// TIA Portal project "Проект3" (V14)

(* hardware
DEVICE "S7300/ET200M station_1"  S7-300 station
   slot 0: "Профильная шина_0"  Rail  6ES7 390-1***0-0AA0
   slot 2: "PLC_1"  CPU 315-2 PN/DP  6ES7 315-2EH14-0AB0  V3.2
      slot 2: "Интерфейс PROFINET_1"  PN-IO
         slot 1: "Порт_1"  Port
         slot 2: "Порт_2"  Port
   slot 4: "DI 32x24 В пост. тока_1"  DI32 x 24VDC  6ES7 321-1BL00-0AA0
   slot 5: "DO 16x24 В пост. тока/0,5 А_1"  DO16 x 24VDC / 0.5A  6ES7 322-1BH01-0AA0
   slot 6: "AI 8x12 бит_1"  AI8 x 12 bits  6ES7 331-7KF02-0AB0
*)

// ===== PLC "PLC_1"  CPU 315-2 PN/DP =====

VAR_GLOBAL   // PLC tag table "Стандартная таблица переменных"
   "Input_1" AT %I0.0 : Bool;
   "Input_2" AT %I0.1 : Bool;
   "Input_3" AT %I0.2 : Bool;
   "Input_4" AT %I0.3 : Bool;
   "Input_5" AT %I0.4 : Bool;
   "Input_6" AT %I0.5 : Bool;
   "Input_7" AT %I0.6 : Bool;
   "Input_8" AT %I0.7 : Bool;
   "Input_9" AT %I1.0 : Bool;
   "Input_10" AT %I1.1 : Bool;
   "Input_11" AT %I1.2 : Bool;
   "Input_12" AT %I1.3 : Bool;
   "Input_13" AT %I1.4 : Bool;
   "Input_14" AT %I1.5 : Bool;
   "Input_15" AT %I1.6 : Bool;
   "Input_16" AT %I1.7 : Bool;
   "Output_1" AT %Q4.0 : Bool;
   "Output_2" AT %Q4.1 : Bool;
   "Output_3" AT %Q4.2 : Bool;
   "Output_4" AT %Q4.3 : Bool;
   "Output_5" AT %Q4.4 : Bool;
   "Output_6" AT %Q4.5 : Bool;
   "Output_7" AT %Q4.6 : Bool;
   "Output_8" AT %Q4.7 : Bool;
   "Output_9" AT %Q5.0 : Bool;
   "Output_10" AT %Q5.1 : Bool;
   "Output_11" AT %Q5.2 : Bool;
   "Output_12" AT %Q5.3 : Bool;
   "Output_13" AT %Q5.4 : Bool;
   "Output_14" AT %Q5.5 : Bool;
   "Output_15" AT %Q5.6 : Bool;
   "Output_16" AT %Q5.7 : Bool;
   "Tag_1" AT %IW0 : Word;
   "Tag_2" AT %IB0 : Byte;
   "Tag_3" AT %IB1 : Byte;
   "Tag_4" AT %QB4 : Byte;
   "Tag_5" AT %QB5 : Byte;
   "Tag_6" AT %IW288 : Int;
   "Tag_7" AT %M0.1 : Bool;
   "Tag_8" AT %MW1 : Word;
   "Tag_9" AT %MW3 : Word;
   "Tag_10" AT %MD4 : Real;
   "Tag_11" AT %IW290 : Int;
   "Tag_12" AT %IW292 : Int;
   "Tag_13" AT %MW10 : Int;
   "Tag_14" AT %MD20 : Real;
   "Tag_15" AT %MW40 : Word;
   "Tag_16" AT %M0.0 : Bool;
   "Tag_17" AT %IW296 : Int;
   "Tag_18" AT %IW298 : Int;
   "Tag_19" AT %MD30 : Real;
   "Tag_20" AT %QD0 : Real;
END_VAR

DATA_BLOCK "DB_1"   // DB1
{ S7_Optimized_Access := 'FALSE' }
VERSION : 0.1
   VAR
      "Q4.0" : Bool;
      "Q4.1" : Bool;
      "Q4.2" : Bool;
      "Q4.3" : Bool;
      "Q4.4" : Bool;
      "Q4.5" : Bool;
      "Q4.6" : Bool;
      "Q4.7" : Bool;
      "Q5.0" : Bool;
      "Q5.1" : Bool;
      "Q5.2" : Bool;
      "Q5.3" : Bool;
      "Q5.4" : Bool;
      "Q5.5" : Bool;
      "Q5.6" : Bool;
      "Q5.7" : Bool;
   END_VAR
BEGIN
END_DATA_BLOCK

DATA_BLOCK "DB_2"   // DB2
{ S7_Optimized_Access := 'FALSE' }
VERSION : 0.1
   VAR
      "i0.0" : Bool;
      "i0.1" : Bool;
      "i0.2" : Bool;
      "i0.3" : Bool;
      "i0.4" : Bool;
      "i0.5" : Bool;
      "i0.6" : Bool;
      "i0.7" : Bool;
      "i1.0" : Bool;
      "i1.1" : Bool;
      "i1.2" : Bool;
      "i1.3" : Bool;
      "i1.4" : Bool;
      "i1.5" : Bool;
      "i1.6" : Bool;
      "i1.7" : Bool;
      md4 : Real;
   END_VAR
BEGIN
END_DATA_BLOCK

ORGANIZATION_BLOCK "Main"   // OB1, LAD
TITLE = "Main Program Sweep (Cycle)"
{ S7_Optimized_Access := 'FALSE' }
VERSION : 0.1
   VAR_TEMP
      OB1_EV_CLASS : Byte;   // Bits 0-3 = 1 (Coming event), Bits 4-7 = 1 (Event class 1)
      OB1_SCAN_1 : Byte;   // 1 (Cold restart scan 1 of OB 1), 3 (Scan 2-n of OB 1)
      OB1_PRIORITY : Byte;   // Priority of OB Execution
      OB1_OB_NUMBR : Byte;   // 1 (Organization block 1, OB1)
      OB1_RESERVED_1 : Byte;   // Reserved for system
      OB1_RESERVED_2 : Byte;   // Reserved for system
      OB1_PREV_CYCLE : Int;   // Cycle time of previous OB1 scan (milliseconds)
      OB1_MIN_CYCLE : Int;   // Minimum cycle time of OB1 (milliseconds)
      OB1_MAX_CYCLE : Int;   // Maximum cycle time of OB1 (milliseconds)
      OB1_DATE_TIME : Date_And_Time;   // Date and time OB1 started
   END_VAR
BEGIN

REGION Network 1
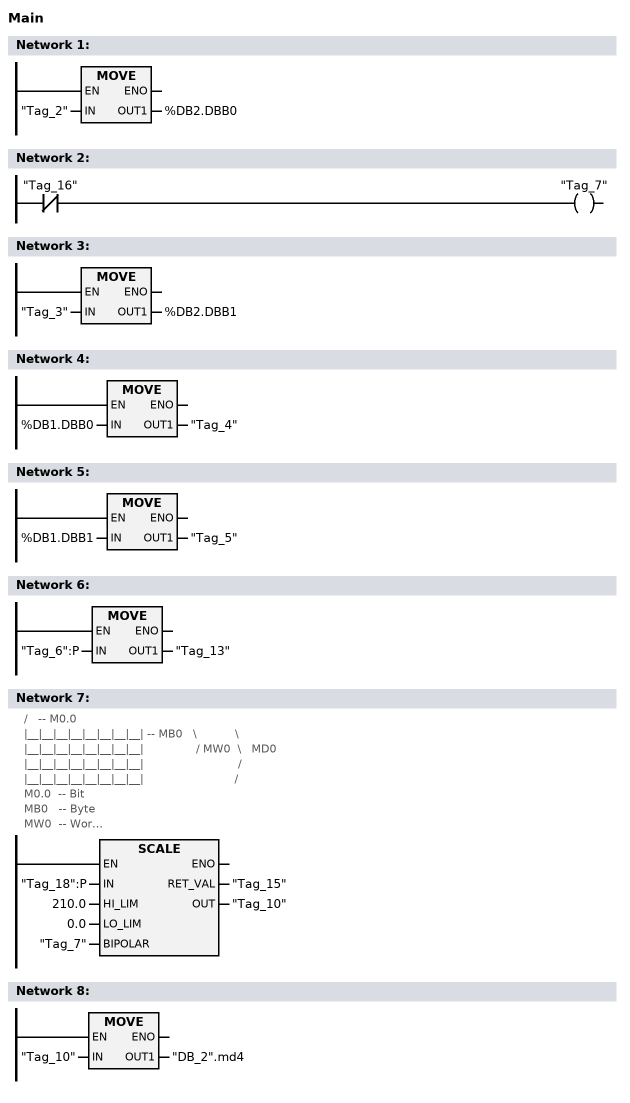
   RUNG wire#powerrail
      { S7_GenerateENO := "TRUE" } Move(in := "Tag_2", out1 => %DB2.DBB0)
   END_RUNG
   // the same network as SCL:
   %DB2.DBB0 := "Tag_2";
END_REGION

REGION Network 2
   RUNG wire#powerrail
      I_Contact( "Tag_16" )
      Coil( "Tag_7" )
   END_RUNG
   // the same network as SCL:
   "Tag_7" := NOT "Tag_16";
END_REGION

REGION Network 3
   RUNG wire#powerrail
      { S7_GenerateENO := "TRUE" } Move(in := "Tag_3", out1 => %DB2.DBB1)
   END_RUNG
   // the same network as SCL:
   %DB2.DBB1 := "Tag_3";
END_REGION

REGION Network 4
   RUNG wire#powerrail
      { S7_GenerateENO := "TRUE" } Move(in := %DB1.DBB0, out1 => "Tag_4")
   END_RUNG
   // the same network as SCL:
   "Tag_4" := %DB1.DBB0;
END_REGION

REGION Network 5
   RUNG wire#powerrail
      { S7_GenerateENO := "TRUE" } Move(in := %DB1.DBB1, out1 => "Tag_5")
   END_RUNG
   // the same network as SCL:
   "Tag_5" := %DB1.DBB1;
END_REGION

REGION Network 6
   RUNG wire#powerrail
      { S7_GenerateENO := "TRUE" } Move(in := "Tag_6":P, out1 => "Tag_13")
   END_RUNG
   // the same network as SCL:
   "Tag_13" := "Tag_6":P;
END_REGION

REGION Network 7
   // /   -- M0.0
   // |__|__|__|__|__|__|__|__| -- MB0   \           \
   // |__|__|__|__|__|__|__|__|               / MW0  \   MD0
   // |__|__|__|__|__|__|__|__|                           /
   // |__|__|__|__|__|__|__|__|                          /
   // 
   // M0.0  -- Bit
   // MB0   -- Byte
   // MW0  -- Word
   // MD0  -- Real
   "Tag_15" := SCALE(IN := "Tag_18":P, HI_LIM := 210.0, LO_LIM := 0.0, BIPOLAR := "Tag_7", OUT => "Tag_10");
END_REGION

REGION Network 8
   RUNG wire#powerrail
      { S7_GenerateENO := "TRUE" } Move(in := "Tag_10", out1 => "DB_2".md4)
   END_RUNG
   // the same network as SCL:
   "DB_2".md4 := "Tag_10";
END_REGION
END_ORGANIZATION_BLOCK